FUNCTION_BLOCK HoldingBitSV
VAR_INPUT

	bSensorRs:BOOL;
	bSv:BOOL;
	bCancelHold:BOOL;

END_VAR
VAR_OUTPUT

	bHoldingBit:BOOL;

END_VAR
VAR
	SensorComfirm: R_TRIG;
END_VAR

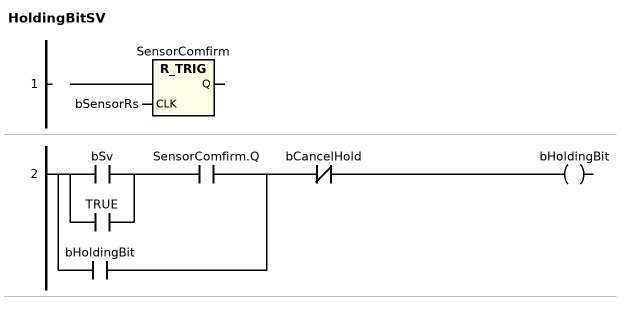
// NETWORK 1
SensorComfirm(CLK := bSensorRs); // R_TRIG

// NETWORK 2
bHoldingBit := ((bSv OR TRUE) AND SensorComfirm.Q OR bHoldingBit) AND NOT bCancelHold;

END_FUNCTION_BLOCK

(* stored: Version 1.1.0.1, ProductVersion 3.1.4024.12
   POU HoldingBitSV: Id {a14e2b9e-4453-4907-a8b5-224ff99ec76a}, SpecialFunc None *)
